Staubli VAL3: cycle_isFound.pgx

program cycle_isFound(string x_sProgName (dimensions=1), bool& x_bFound[] (dimensions=1))
  local num i
begin
  x_bFound=false
  // verify if a program is in the program list
  // libList(saveData:sPathProg[0],sProgList)
  // check inside the program List
  for i=0 to size(sProgList)-1
    if sProgList[min(size(sProgList)-1,i)]==x_sProgName
      x_bFound=true
      return
    endIf
  endFor
end
